// TIA Portal V20 export
FUNCTION "LER_Axis64PosCommand" : Void   // FC93, LAD
// stored: Access Published, SetENOAutomatically false
   VAR_INPUT
      enable : Bool;
   END_VAR
   VAR_IN_OUT
      Command : USInt;
      Axis64PosControl : "LBC_typeAxis64PosControlNode";
   END_VAR
   VAR CONSTANT
      CommandReset : USInt;
      CommandMoveVelocity : USInt := 1;
      CommandTorqueLimiting : USInt := 2;
      CommandHoming : USInt := 3;
      CommandPosRelative : USInt := 4;
      CommandposAbsolute : USInt := 5;
      CommandposSuperimposed : USInt := 6;
      CommandHalt : USInt := 7;
      CommandGearIn : USInt := 8;
      CommandCamIn : USInt := 9;
      CommandGearOutCamOut : USInt := 10;
      CommandPhasing : USInt := 11;
   END_VAR
BEGIN

REGION Network 1: Rising edge: Move an axis at constant velocity/speed
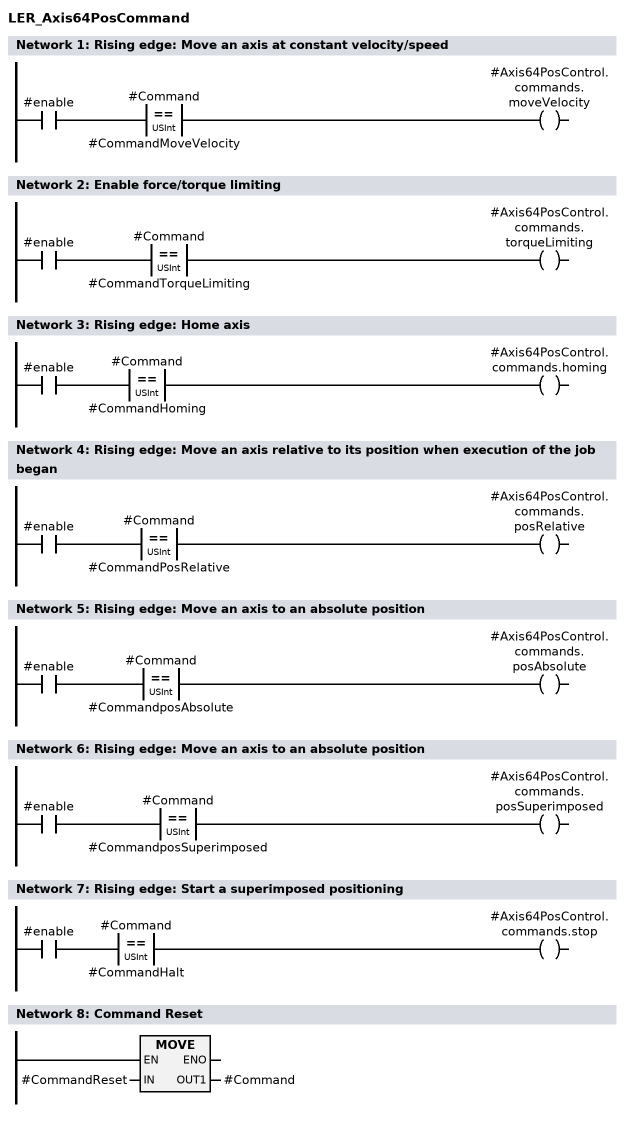
   RUNG wire#powerrail
      Contact( #enable )
      { S7_Templates := "SrcType := USInt" } EQ_Contact(in1 := #Command, in2 := #CommandMoveVelocity)
      Coil( #Axis64PosControl.commands.moveVelocity )
   END_RUNG
   // the same network as SCL:
   #Axis64PosControl.commands.moveVelocity := #enable AND (#Command = #CommandMoveVelocity);
END_REGION

REGION Network 2: Enable force/torque limiting
   RUNG wire#powerrail
      Contact( #enable )
      { S7_Templates := "SrcType := USInt" } EQ_Contact(in1 := #Command, in2 := #CommandTorqueLimiting)
      Coil( #Axis64PosControl.commands.torqueLimiting )
   END_RUNG
   // the same network as SCL:
   #Axis64PosControl.commands.torqueLimiting := #enable AND (#Command = #CommandTorqueLimiting);
END_REGION

REGION Network 3: Rising edge: Home axis
   RUNG wire#powerrail
      Contact( #enable )
      { S7_Templates := "SrcType := USInt" } EQ_Contact(in1 := #Command, in2 := #CommandHoming)
      Coil( #Axis64PosControl.commands.homing )
   END_RUNG
   // the same network as SCL:
   #Axis64PosControl.commands.homing := #enable AND (#Command = #CommandHoming);
END_REGION

REGION Network 4: Rising edge: Move an axis relative to its position when execution of the job began
   RUNG wire#powerrail
      Contact( #enable )
      { S7_Templates := "SrcType := USInt" } EQ_Contact(in1 := #Command, in2 := #CommandPosRelative)
      Coil( #Axis64PosControl.commands.posRelative )
   END_RUNG
   // the same network as SCL:
   #Axis64PosControl.commands.posRelative := #enable AND (#Command = #CommandPosRelative);
END_REGION

REGION Network 5: Rising edge: Move an axis to an absolute position
   RUNG wire#powerrail
      Contact( #enable )
      { S7_Templates := "SrcType := USInt" } EQ_Contact(in1 := #Command, in2 := #CommandposAbsolute)
      Coil( #Axis64PosControl.commands.posAbsolute )
   END_RUNG
   // the same network as SCL:
   #Axis64PosControl.commands.posAbsolute := #enable AND (#Command = #CommandposAbsolute);
END_REGION

REGION Network 6: Rising edge: Move an axis to an absolute position
   RUNG wire#powerrail
      Contact( #enable )
      { S7_Templates := "SrcType := USInt" } EQ_Contact(in1 := #Command, in2 := #CommandposSuperimposed)
      Coil( #Axis64PosControl.commands.posSuperimposed )
   END_RUNG
   // the same network as SCL:
   #Axis64PosControl.commands.posSuperimposed := #enable AND (#Command = #CommandposSuperimposed);
END_REGION

REGION Network 7: Rising edge: Start a superimposed positioning
   RUNG wire#powerrail
      Contact( #enable )
      { S7_Templates := "SrcType := USInt" } EQ_Contact(in1 := #Command, in2 := #CommandHalt)
      Coil( #Axis64PosControl.commands.stop )
   END_RUNG
   // the same network as SCL:
   #Axis64PosControl.commands.stop := #enable AND (#Command = #CommandHalt);
END_REGION

REGION Network 8: Command Reset
   RUNG wire#powerrail
      Move(in := #CommandReset, out1 => #Command)
   END_RUNG
   // the same network as SCL:
   #Command := #CommandReset;
END_REGION
END_FUNCTION
